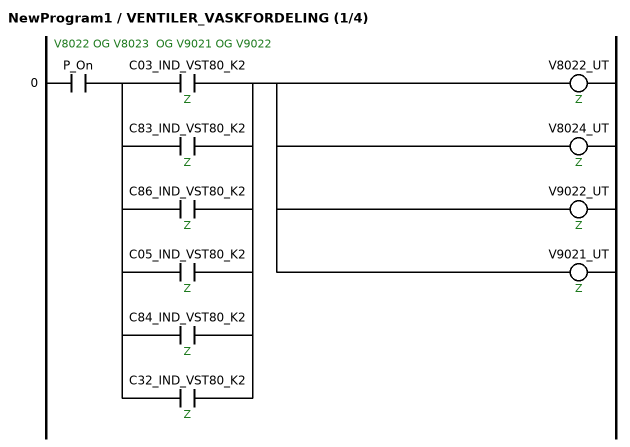
; [picture p840: NewProgram1 / VENTILER_VASKFORDELING, rungs 0-0]
; rung 0: V8022 OG V8023  OG V9021 OG V9022
LD P_On
LD C03_IND_VST80_K2  ; Z
OR C83_IND_VST80_K2  ; Z
OR C86_IND_VST80_K2  ; Z
OR C05_IND_VST80_K2  ; Z
OR C84_IND_VST80_K2  ; Z
OR C32_IND_VST80_K2  ; Z
ANDLD
OUT V8022_UT  ; Z
OUT V8024_UT  ; Z
OUT V9022_UT  ; Z
OUT V9021_UT  ; Z

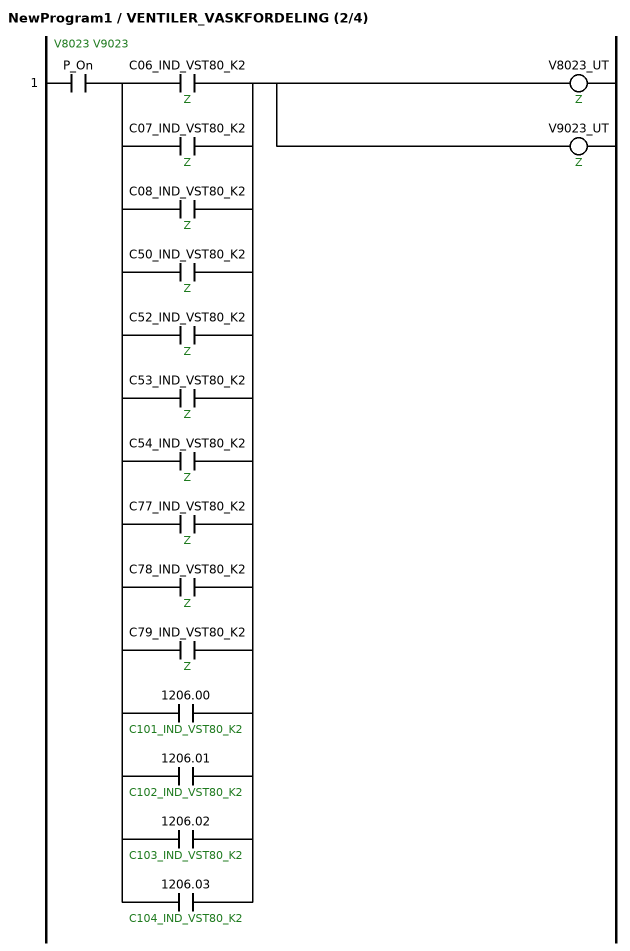
; rung 1: V8023 V9023
LD P_On
LD C06_IND_VST80_K2  ; Z
OR C07_IND_VST80_K2  ; Z
OR C08_IND_VST80_K2  ; Z
OR C50_IND_VST80_K2  ; Z
OR C52_IND_VST80_K2  ; Z
OR C53_IND_VST80_K2  ; Z
OR C54_IND_VST80_K2  ; Z
OR C77_IND_VST80_K2  ; Z
OR C78_IND_VST80_K2  ; Z
OR C79_IND_VST80_K2  ; Z
OR 1206.00  ; C101_IND_VST80_K2
OR 1206.01  ; C102_IND_VST80_K2
OR 1206.02  ; C103_IND_VST80_K2
OR 1206.03  ; C104_IND_VST80_K2
ANDLD
OUT V8023_UT  ; Z
OUT V9023_UT  ; Z

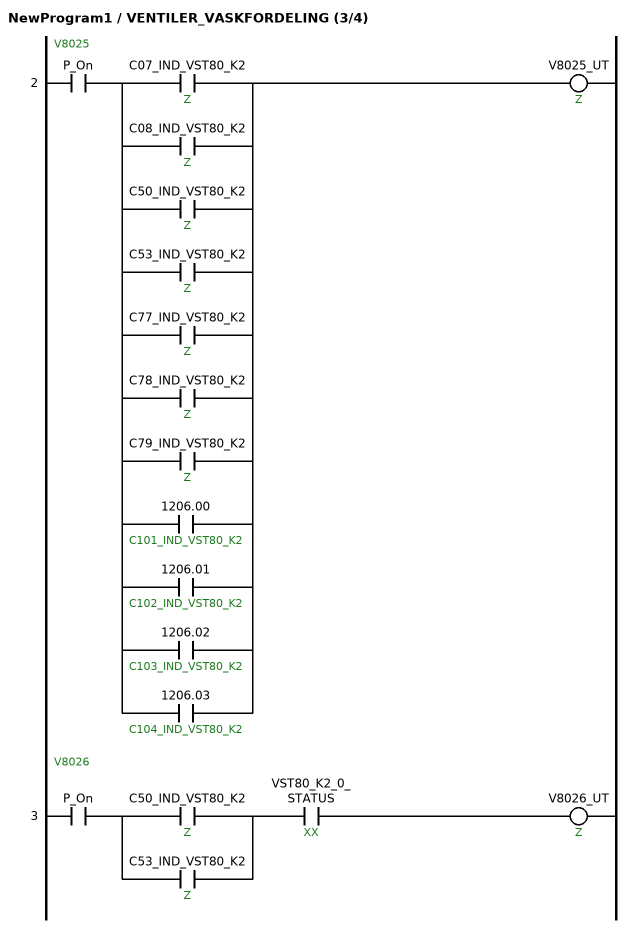
; rung 2: V8025
LD P_On
LD C07_IND_VST80_K2  ; Z
OR C08_IND_VST80_K2  ; Z
OR C50_IND_VST80_K2  ; Z
OR C53_IND_VST80_K2  ; Z
OR C77_IND_VST80_K2  ; Z
OR C78_IND_VST80_K2  ; Z
OR C79_IND_VST80_K2  ; Z
OR 1206.00  ; C101_IND_VST80_K2
OR 1206.01  ; C102_IND_VST80_K2
OR 1206.02  ; C103_IND_VST80_K2
OR 1206.03  ; C104_IND_VST80_K2
ANDLD
OUT V8025_UT  ; Z
; rung 3: V8026
LD P_On
LD C50_IND_VST80_K2  ; Z
OR C53_IND_VST80_K2  ; Z
ANDLD
AND VST80_K2_0_STATUS  ; XX
OUT V8026_UT  ; Z

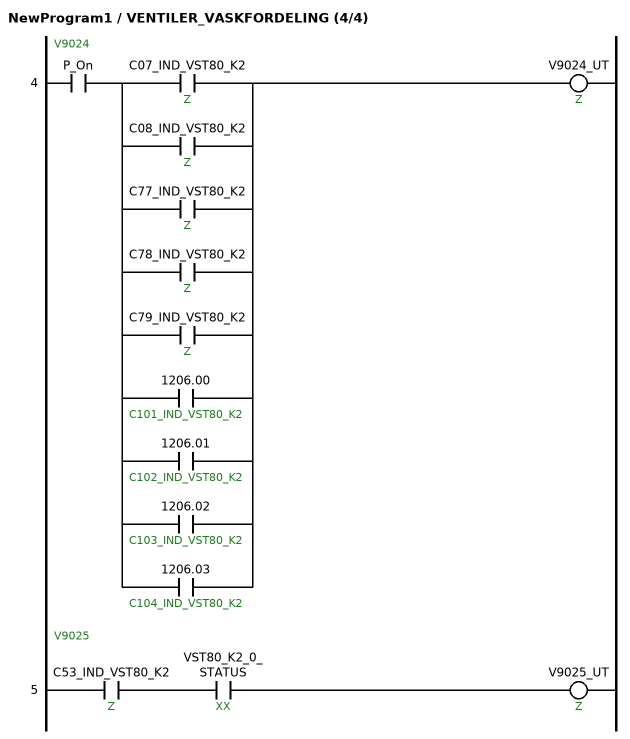
; rung 4: V9024
LD P_On
LD C07_IND_VST80_K2  ; Z
OR C08_IND_VST80_K2  ; Z
OR C77_IND_VST80_K2  ; Z
OR C78_IND_VST80_K2  ; Z
OR C79_IND_VST80_K2  ; Z
OR 1206.00  ; C101_IND_VST80_K2
OR 1206.01  ; C102_IND_VST80_K2
OR 1206.02  ; C103_IND_VST80_K2
OR 1206.03  ; C104_IND_VST80_K2
ANDLD
OUT V9024_UT  ; Z
; rung 5: V9025
LD C53_IND_VST80_K2  ; Z
AND VST80_K2_0_STATUS  ; XX
OUT V9025_UT  ; Z
; rung 6: Ingen_kommentar_funnet

### Section VENTILER_BILVASK

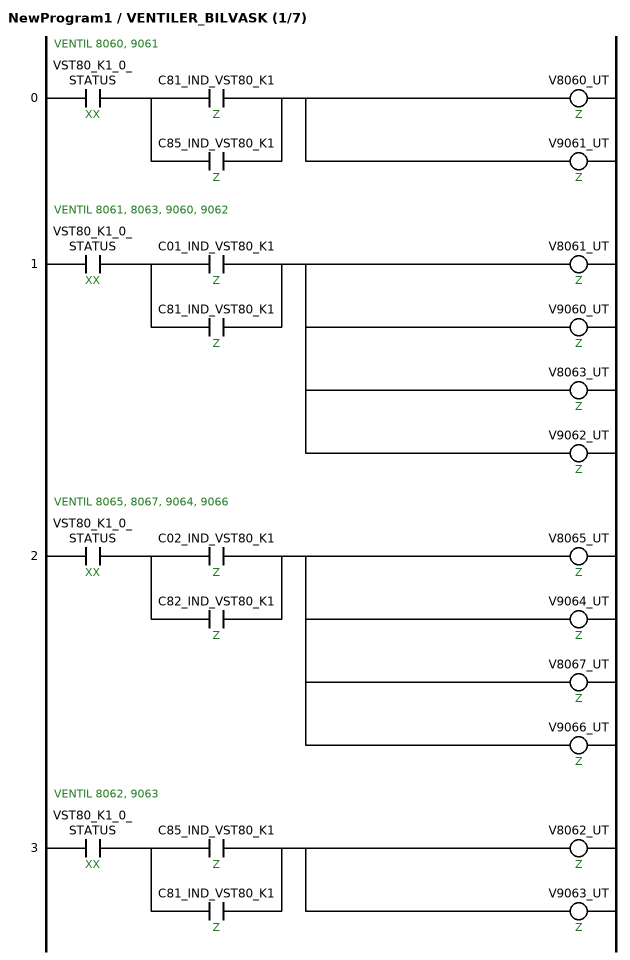
; rung 0: VENTIL 8060, 9061
LD VST80_K1_0_STATUS  ; XX
LD C81_IND_VST80_K1  ; Z
OR C85_IND_VST80_K1  ; Z
ANDLD
OUT V8060_UT  ; Z
OUT V9061_UT  ; Z
; rung 1: VENTIL 8061, 8063, 9060, 9062
LD VST80_K1_0_STATUS  ; XX
LD C01_IND_VST80_K1  ; Z
OR C81_IND_VST80_K1  ; Z
ANDLD
OUT V8061_UT  ; Z
OUT V9060_UT  ; Z
OUT V8063_UT  ; Z
OUT V9062_UT  ; Z
; rung 2: VENTIL 8065, 8067, 9064, 9066
LD VST80_K1_0_STATUS  ; XX
LD C02_IND_VST80_K1  ; Z
OR C82_IND_VST80_K1  ; Z
ANDLD
OUT V8065_UT  ; Z
OUT V9064_UT  ; Z
OUT V8067_UT  ; Z
OUT V9066_UT  ; Z
; rung 3: VENTIL 8062, 9063
LD VST80_K1_0_STATUS  ; XX
LD C85_IND_VST80_K1  ; Z
OR C81_IND_VST80_K1  ; Z
ANDLD
OUT V8062_UT  ; Z
OUT V9063_UT  ; Z

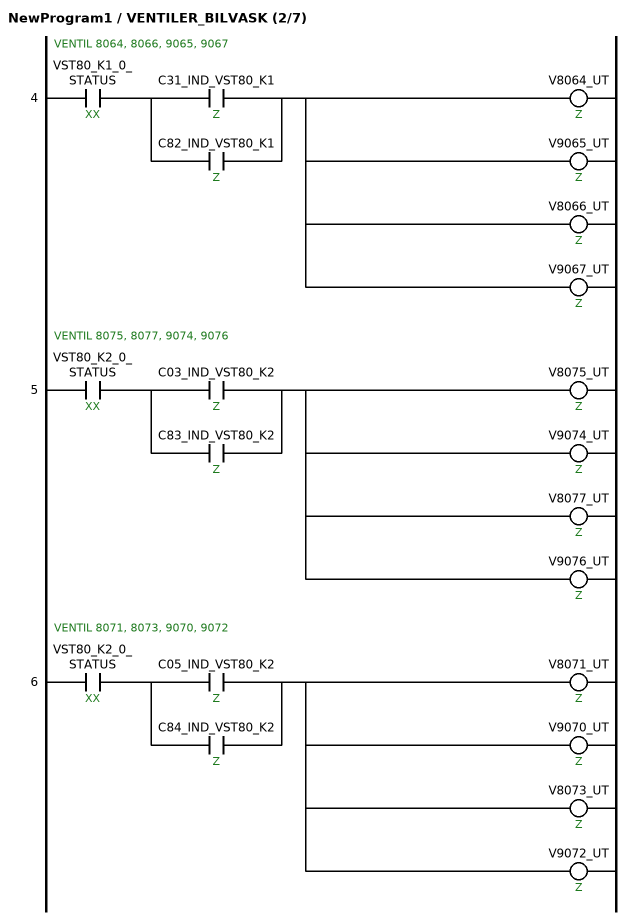
; rung 4: VENTIL 8064, 8066, 9065, 9067
LD VST80_K1_0_STATUS  ; XX
LD C31_IND_VST80_K1  ; Z
OR C82_IND_VST80_K1  ; Z
ANDLD
OUT V8064_UT  ; Z
OUT V9065_UT  ; Z
OUT V8066_UT  ; Z
OUT V9067_UT  ; Z
; rung 5: VENTIL 8075, 8077, 9074, 9076
LD VST80_K2_0_STATUS  ; XX
LD C03_IND_VST80_K2  ; Z
OR C83_IND_VST80_K2  ; Z
ANDLD
OUT V8075_UT  ; Z
OUT V9074_UT  ; Z
OUT V8077_UT  ; Z
OUT V9076_UT  ; Z
; rung 6: VENTIL 8071, 8073, 9070, 9072
LD VST80_K2_0_STATUS  ; XX
LD C05_IND_VST80_K2  ; Z
OR C84_IND_VST80_K2  ; Z
ANDLD
OUT V8071_UT  ; Z
OUT V9070_UT  ; Z
OUT V8073_UT  ; Z
OUT V9072_UT  ; Z

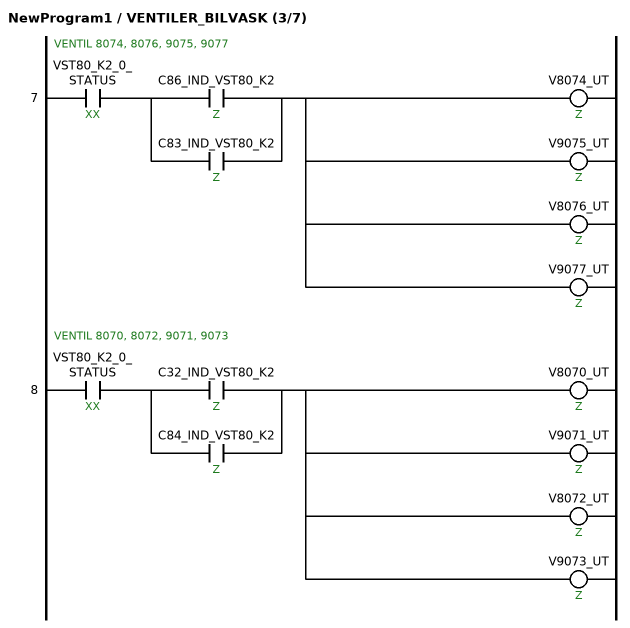
; rung 7: VENTIL 8074, 8076, 9075, 9077
LD VST80_K2_0_STATUS  ; XX
LD C86_IND_VST80_K2  ; Z
OR C83_IND_VST80_K2  ; Z
ANDLD
OUT V8074_UT  ; Z
OUT V9075_UT  ; Z
OUT V8076_UT  ; Z
OUT V9077_UT  ; Z
; rung 8: VENTIL 8070, 8072, 9071, 9073
LD VST80_K2_0_STATUS  ; XX
LD C32_IND_VST80_K2  ; Z
OR C84_IND_VST80_K2  ; Z
ANDLD
OUT V8070_UT  ; Z
OUT V9071_UT  ; Z
OUT V8072_UT  ; Z
OUT V9073_UT  ; Z

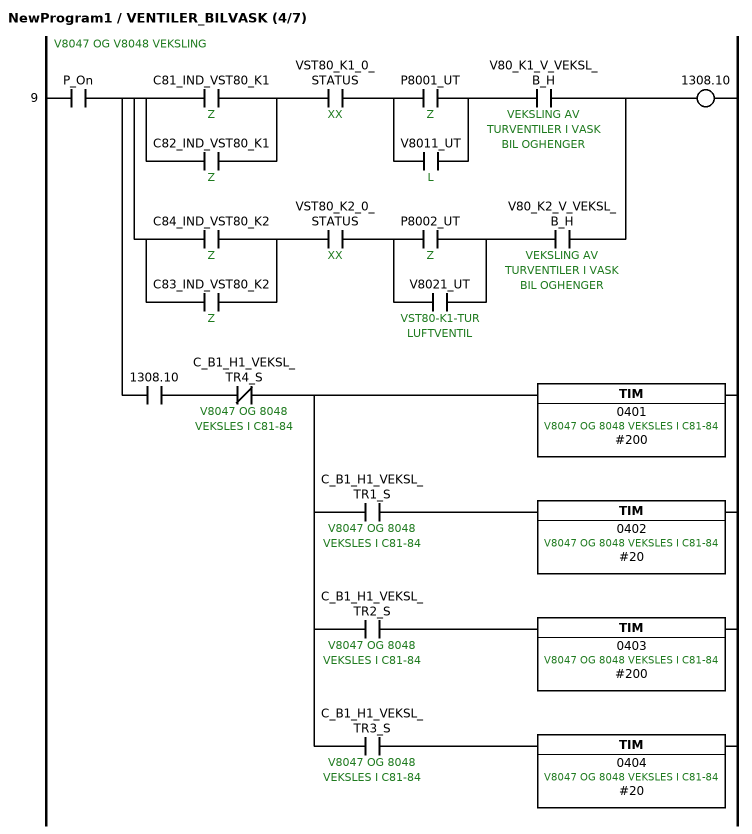
; rung 9: V8047 OG V8048 VEKSLING
LD P_On
OUT TR0
LD C81_IND_VST80_K1  ; Z
OR C82_IND_VST80_K1  ; Z
AND VST80_K1_0_STATUS  ; XX
LD P8001_UT  ; Z
OR V8011_UT  ; L
ANDLD
AND V80_K1_V_VEKSL_B_H  ; VEKSLING AV TURVENTILER I VASK BIL OGHENGER
LD C84_IND_VST80_K2  ; Z
OR C83_IND_VST80_K2  ; Z
AND VST80_K2_0_STATUS  ; XX
LD P8002_UT  ; Z
OR V8021_UT  ; VST80-K1-TUR LUFTVENTIL
ANDLD
AND V80_K2_V_VEKSL_B_H  ; VEKSLING AV TURVENTILER I VASK BIL OGHENGER
ORLD
ANDLD
OUT 1308.10
LD TR0
AND 1308.10
ANDNOT C_B1_H1_VEKSL_TR4_S  ; V8047 OG 8048 VEKSLES I C81-84
OUT TR0
TIM 0401 #200  ; V8047 OG 8048 VEKSLES I C81-84
AND C_B1_H1_VEKSL_TR1_S  ; V8047 OG 8048 VEKSLES I C81-84
TIM 0402 #20  ; V8047 OG 8048 VEKSLES I C81-84
LD TR0
AND C_B1_H1_VEKSL_TR2_S  ; V8047 OG 8048 VEKSLES I C81-84
TIM 0403 #200  ; V8047 OG 8048 VEKSLES I C81-84
LD TR0
AND C_B1_H1_VEKSL_TR3_S  ; V8047 OG 8048 VEKSLES I C81-84
TIM 0404 #20  ; V8047 OG 8048 VEKSLES I C81-84

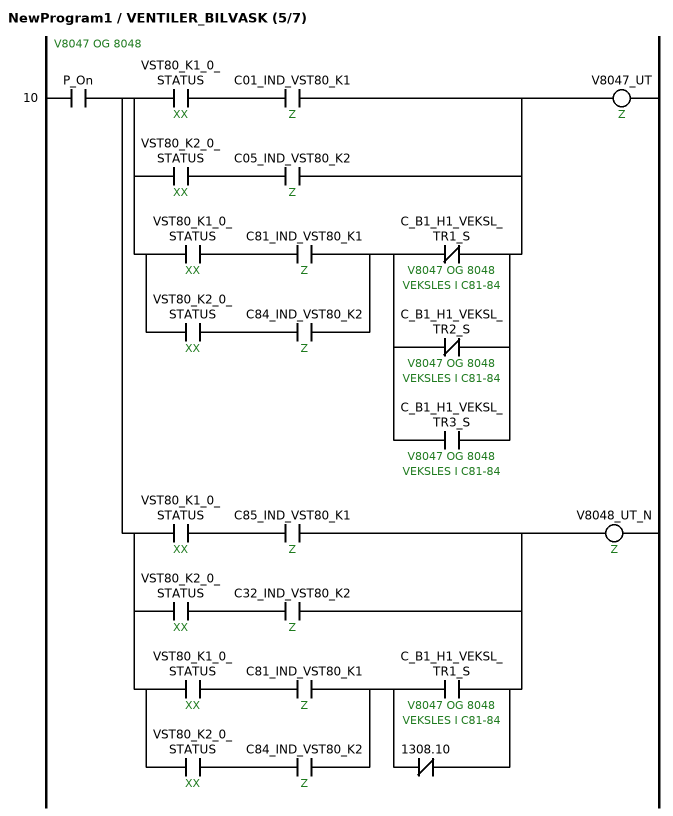
; rung 10: V8047 OG 8048
LD P_On
OUT TR0
LD VST80_K1_0_STATUS  ; XX
AND C01_IND_VST80_K1  ; Z
LD VST80_K2_0_STATUS  ; XX
AND C05_IND_VST80_K2  ; Z
ORLD
LD VST80_K1_0_STATUS  ; XX
AND C81_IND_VST80_K1  ; Z
LD VST80_K2_0_STATUS  ; XX
AND C84_IND_VST80_K2  ; Z
ORLD
LDNOT C_B1_H1_VEKSL_TR1_S  ; V8047 OG 8048 VEKSLES I C81-84
ORNOT C_B1_H1_VEKSL_TR2_S  ; V8047 OG 8048 VEKSLES I C81-84
OR C_B1_H1_VEKSL_TR3_S  ; V8047 OG 8048 VEKSLES I C81-84
ANDLD
ORLD
ANDLD
OUT V8047_UT  ; Z
LD TR0
LD VST80_K1_0_STATUS  ; XX
AND C85_IND_VST80_K1  ; Z
LD VST80_K2_0_STATUS  ; XX
AND C32_IND_VST80_K2  ; Z
ORLD
LD VST80_K1_0_STATUS  ; XX
AND C81_IND_VST80_K1  ; Z
LD VST80_K2_0_STATUS  ; XX
AND C84_IND_VST80_K2  ; Z
ORLD
LD C_B1_H1_VEKSL_TR1_S  ; V8047 OG 8048 VEKSLES I C81-84
ORNOT 1308.10
ANDLD
ORLD
ANDLD
OUT V8048_UT_N  ; Z

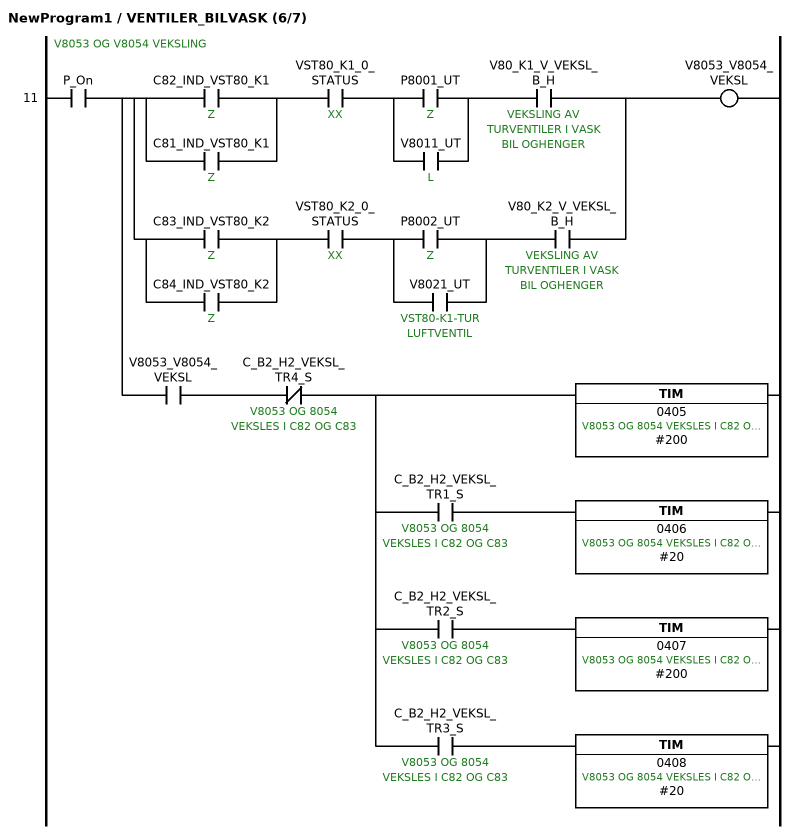
; rung 11: V8053 OG V8054 VEKSLING
LD P_On
OUT TR0
LD C82_IND_VST80_K1  ; Z
OR C81_IND_VST80_K1  ; Z
AND VST80_K1_0_STATUS  ; XX
LD P8001_UT  ; Z
OR V8011_UT  ; L
ANDLD
AND V80_K1_V_VEKSL_B_H  ; VEKSLING AV TURVENTILER I VASK BIL OGHENGER
LD C83_IND_VST80_K2  ; Z
OR C84_IND_VST80_K2  ; Z
AND VST80_K2_0_STATUS  ; XX
LD P8002_UT  ; Z
OR V8021_UT  ; VST80-K1-TUR LUFTVENTIL
ANDLD
AND V80_K2_V_VEKSL_B_H  ; VEKSLING AV TURVENTILER I VASK BIL OGHENGER
ORLD
ANDLD
OUT V8053_V8054_VEKSL
LD TR0
AND V8053_V8054_VEKSL
ANDNOT C_B2_H2_VEKSL_TR4_S  ; V8053 OG 8054 VEKSLES I C82 OG C83
OUT TR0
TIM 0405 #200  ; V8053 OG 8054 VEKSLES I C82 OG C83
AND C_B2_H2_VEKSL_TR1_S  ; V8053 OG 8054 VEKSLES I C82 OG C83
TIM 0406 #20  ; V8053 OG 8054 VEKSLES I C82 OG C83
LD TR0
AND C_B2_H2_VEKSL_TR2_S  ; V8053 OG 8054 VEKSLES I C82 OG C83
TIM 0407 #200  ; V8053 OG 8054 VEKSLES I C82 OG C83
LD TR0
AND C_B2_H2_VEKSL_TR3_S  ; V8053 OG 8054 VEKSLES I C82 OG C83
TIM 0408 #20  ; V8053 OG 8054 VEKSLES I C82 OG C83

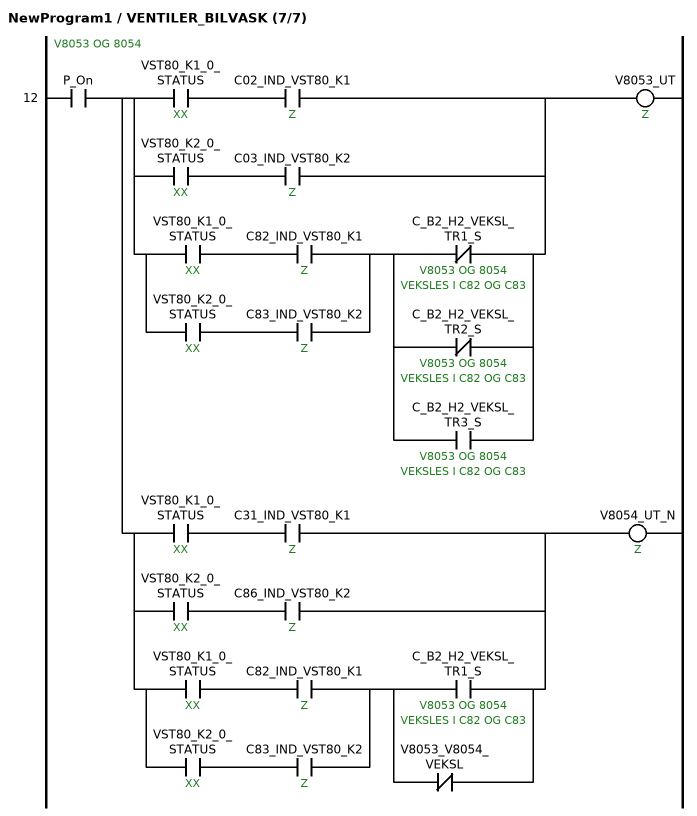
; rung 12: V8053 OG 8054
LD P_On
OUT TR0
LD VST80_K1_0_STATUS  ; XX
AND C02_IND_VST80_K1  ; Z
LD VST80_K2_0_STATUS  ; XX
AND C03_IND_VST80_K2  ; Z
ORLD
LD VST80_K1_0_STATUS  ; XX
AND C82_IND_VST80_K1  ; Z
LD VST80_K2_0_STATUS  ; XX
AND C83_IND_VST80_K2  ; Z
ORLD
LDNOT C_B2_H2_VEKSL_TR1_S  ; V8053 OG 8054 VEKSLES I C82 OG C83
ORNOT C_B2_H2_VEKSL_TR2_S  ; V8053 OG 8054 VEKSLES I C82 OG C83
OR C_B2_H2_VEKSL_TR3_S  ; V8053 OG 8054 VEKSLES I C82 OG C83
ANDLD
ORLD
ANDLD
OUT V8053_UT  ; Z
LD TR0
LD VST80_K1_0_STATUS  ; XX
AND C31_IND_VST80_K1  ; Z
LD VST80_K2_0_STATUS  ; XX
AND C86_IND_VST80_K2  ; Z
ORLD
LD VST80_K1_0_STATUS  ; XX
AND C82_IND_VST80_K1  ; Z
LD VST80_K2_0_STATUS  ; XX
AND C83_IND_VST80_K2  ; Z
ORLD
LD C_B2_H2_VEKSL_TR1_S  ; V8053 OG 8054 VEKSLES I C82 OG C83
ORNOT V8053_V8054_VEKSL
ANDLD
ORLD
ANDLD
OUT V8054_UT_N  ; Z
; rung 13: Ingen_kommentar_funnet

### Section VENTILER_SILOTANKER

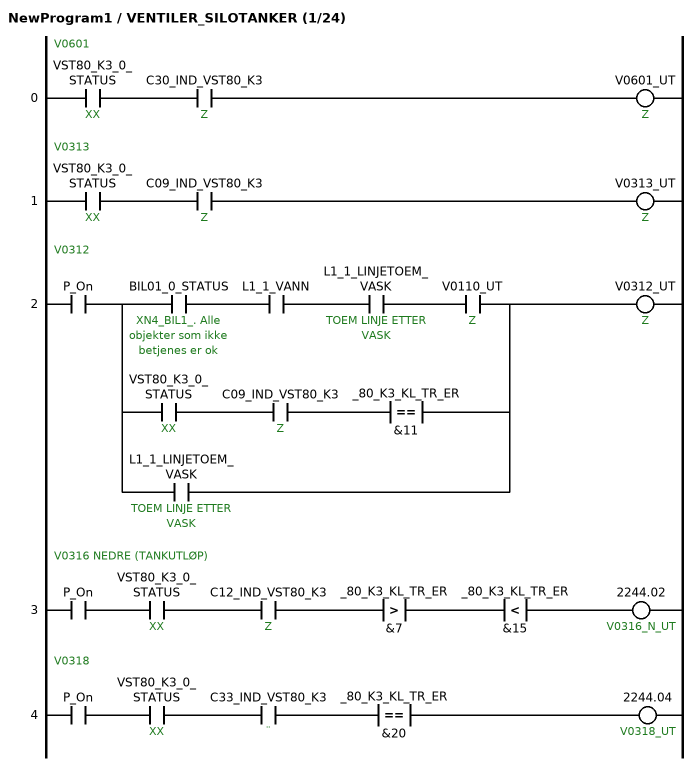
; rung 0: V0601
LD VST80_K3_0_STATUS  ; XX
AND C30_IND_VST80_K3  ; Z
OUT V0601_UT  ; Z
; rung 1: V0313
LD VST80_K3_0_STATUS  ; XX
AND C09_IND_VST80_K3  ; Z
OUT V0313_UT  ; Z
; rung 2: V0312
LD P_On
LD BIL01_0_STATUS  ; XN4_BIL1_. Alle objekter som ikke betjenes er ok
AND L1_1_VANN
AND L1_1_LINJETOEM_VASK  ; TOEM LINJE ETTER VASK
AND V0110_UT  ; Z
LD VST80_K3_0_STATUS  ; XX
AND C09_IND_VST80_K3  ; Z
AND=(300) _80_K3_KL_TR_ER &11
ORLD
OR L1_1_LINJETOEM_VASK  ; TOEM LINJE ETTER VASK
ANDLD
OUT V0312_UT  ; Z
; rung 3: V0316 NEDRE (TANKUTLØP)
LD P_On
AND VST80_K3_0_STATUS  ; XX
AND C12_IND_VST80_K3  ; Z
AND>(320) _80_K3_KL_TR_ER &7
AND<(310) _80_K3_KL_TR_ER &15
OUT 2244.02  ; V0316_N_UT
; rung 4: V0318
LD P_On
AND VST80_K3_0_STATUS  ; XX
AND C33_IND_VST80_K3  ; ¨
AND=(300) _80_K3_KL_TR_ER &20
OUT 2244.04  ; V0318_UT

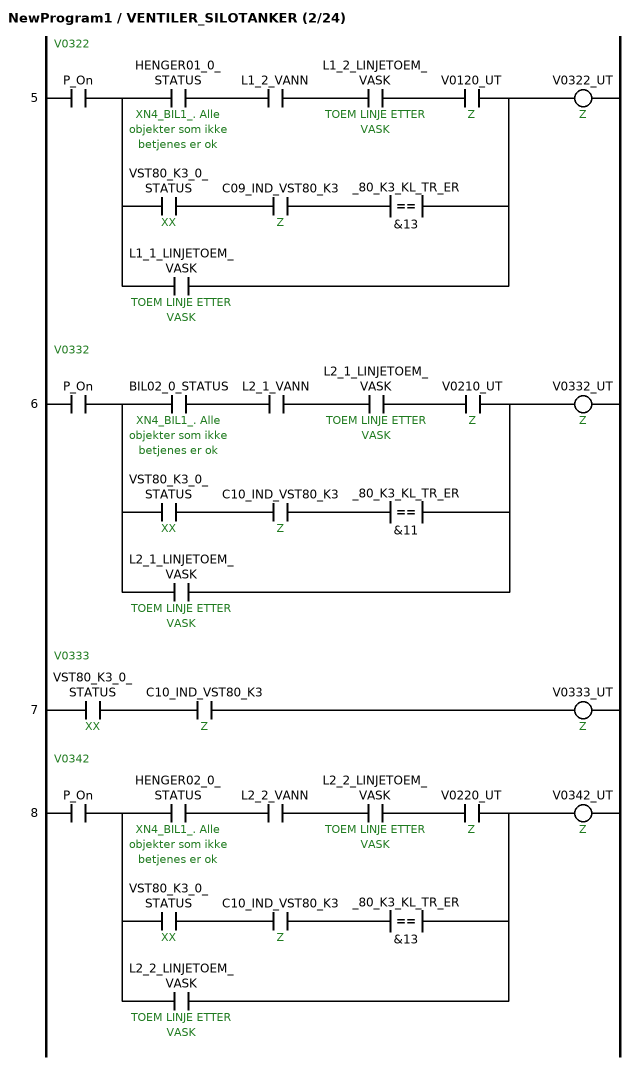
; rung 5: V0322
LD P_On
LD HENGER01_0_STATUS  ; XN4_BIL1_. Alle objekter som ikke betjenes er ok
AND L1_2_VANN
AND L1_2_LINJETOEM_VASK  ; TOEM LINJE ETTER VASK
AND V0120_UT  ; Z
LD VST80_K3_0_STATUS  ; XX
AND C09_IND_VST80_K3  ; Z
AND=(300) _80_K3_KL_TR_ER &13
ORLD
OR L1_1_LINJETOEM_VASK  ; TOEM LINJE ETTER VASK
ANDLD
OUT V0322_UT  ; Z
; rung 6: V0332
LD P_On
LD BIL02_0_STATUS  ; XN4_BIL1_. Alle objekter som ikke betjenes er ok
AND L2_1_VANN
AND L2_1_LINJETOEM_VASK  ; TOEM LINJE ETTER VASK
AND V0210_UT  ; Z
LD VST80_K3_0_STATUS  ; XX
AND C10_IND_VST80_K3  ; Z
AND=(300) _80_K3_KL_TR_ER &11
ORLD
OR L2_1_LINJETOEM_VASK  ; TOEM LINJE ETTER VASK
ANDLD
OUT V0332_UT  ; Z
; rung 7: V0333
LD VST80_K3_0_STATUS  ; XX
AND C10_IND_VST80_K3  ; Z
OUT V0333_UT  ; Z
; rung 8: V0342
LD P_On
LD HENGER02_0_STATUS  ; XN4_BIL1_. Alle objekter som ikke betjenes er ok
AND L2_2_VANN
AND L2_2_LINJETOEM_VASK  ; TOEM LINJE ETTER VASK
AND V0220_UT  ; Z
LD VST80_K3_0_STATUS  ; XX
AND C10_IND_VST80_K3  ; Z
AND=(300) _80_K3_KL_TR_ER &13
ORLD
OR L2_2_LINJETOEM_VASK  ; TOEM LINJE ETTER VASK
ANDLD
OUT V0342_UT  ; Z

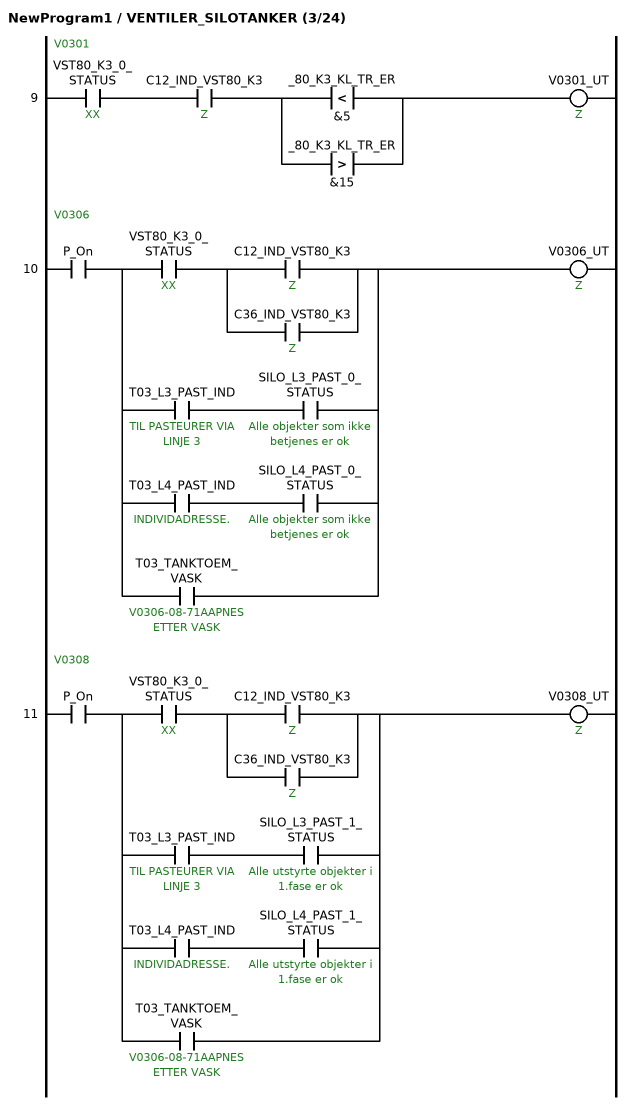
; rung 9: V0301
LD VST80_K3_0_STATUS  ; XX
AND C12_IND_VST80_K3  ; Z
LD<(310) _80_K3_KL_TR_ER &5
OR>(320) _80_K3_KL_TR_ER &15
ANDLD
OUT V0301_UT  ; Z
; rung 10: V0306
LD P_On
LD VST80_K3_0_STATUS  ; XX
LD C12_IND_VST80_K3  ; Z
OR C36_IND_VST80_K3  ; Z
ANDLD
LD T03_L3_PAST_IND  ; TIL PASTEURER VIA LINJE 3
AND SILO_L3_PAST_0_STATUS  ; Alle objekter som ikke betjenes er ok
ORLD
LD T03_L4_PAST_IND  ; INDIVIDADRESSE.
AND SILO_L4_PAST_0_STATUS  ; Alle objekter som ikke betjenes er ok
ORLD
OR T03_TANKTOEM_VASK  ; V0306-08-71AAPNES ETTER VASK
ANDLD
OUT V0306_UT  ; Z
; rung 11: V0308
LD P_On
LD VST80_K3_0_STATUS  ; XX
LD C12_IND_VST80_K3  ; Z
OR C36_IND_VST80_K3  ; Z
ANDLD
LD T03_L3_PAST_IND  ; TIL PASTEURER VIA LINJE 3
AND SILO_L3_PAST_1_STATUS  ; Alle utstyrte objekter i 1.fase er ok
ORLD
LD T03_L4_PAST_IND  ; INDIVIDADRESSE.
AND SILO_L4_PAST_1_STATUS  ; Alle utstyrte objekter i 1.fase er ok
ORLD
OR T03_TANKTOEM_VASK  ; V0306-08-71AAPNES ETTER VASK
ANDLD
OUT V0308_UT  ; Z

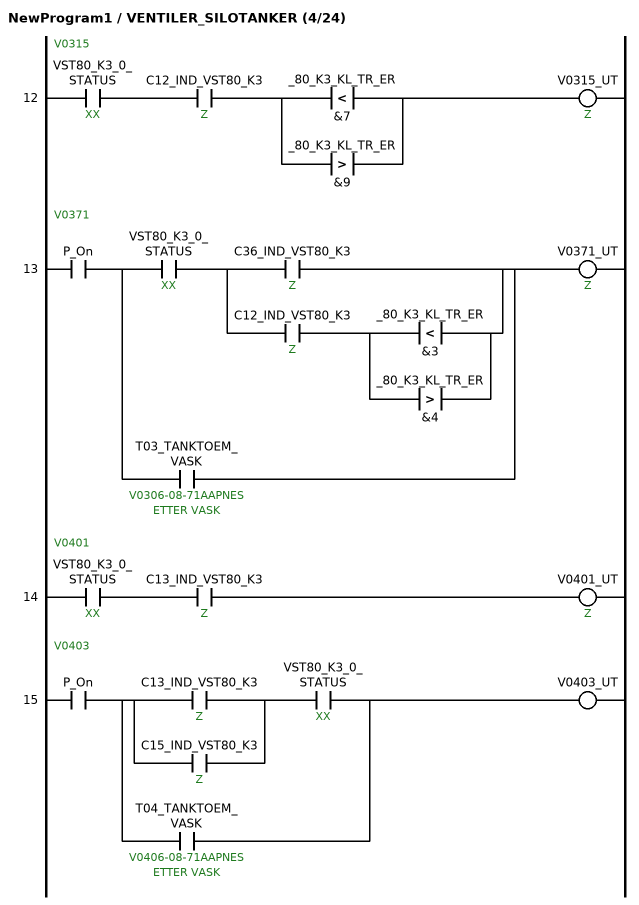
; rung 12: V0315
LD VST80_K3_0_STATUS  ; XX
AND C12_IND_VST80_K3  ; Z
LD<(310) _80_K3_KL_TR_ER &7
OR>(320) _80_K3_KL_TR_ER &9
ANDLD
OUT V0315_UT  ; Z
; rung 13: V0371
LD P_On
LD VST80_K3_0_STATUS  ; XX
LD C36_IND_VST80_K3  ; Z
LD C12_IND_VST80_K3  ; Z
LD<(310) _80_K3_KL_TR_ER &3
OR>(320) _80_K3_KL_TR_ER &4
ANDLD
ORLD
ANDLD
OR T03_TANKTOEM_VASK  ; V0306-08-71AAPNES ETTER VASK
ANDLD
OUT V0371_UT  ; Z
; rung 14: V0401
LD VST80_K3_0_STATUS  ; XX
AND C13_IND_VST80_K3  ; Z
OUT V0401_UT  ; Z
; rung 15: V0403
LD P_On
LD C13_IND_VST80_K3  ; Z
OR C15_IND_VST80_K3  ; Z
AND VST80_K3_0_STATUS  ; XX
OR T04_TANKTOEM_VASK  ; V0406-08-71AAPNES ETTER VASK
ANDLD
OUT V0403_UT

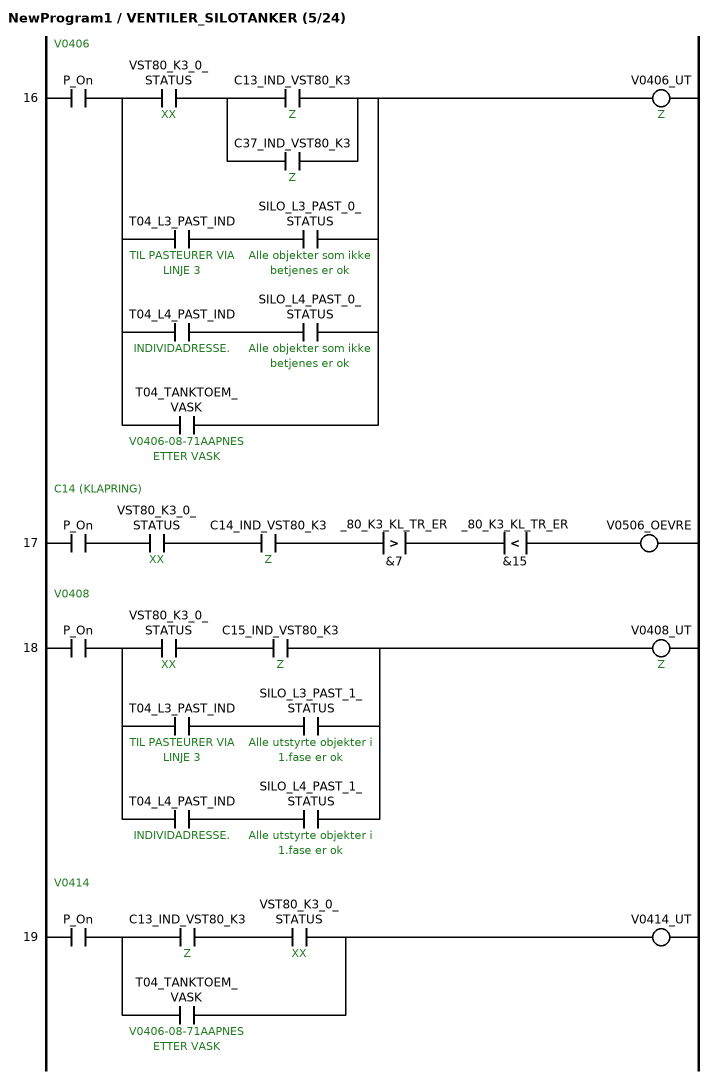
; rung 16: V0406
LD P_On
LD VST80_K3_0_STATUS  ; XX
LD C13_IND_VST80_K3  ; Z
OR C37_IND_VST80_K3  ; Z
ANDLD
LD T04_L3_PAST_IND  ; TIL PASTEURER VIA LINJE 3
AND SILO_L3_PAST_0_STATUS  ; Alle objekter som ikke betjenes er ok
ORLD
LD T04_L4_PAST_IND  ; INDIVIDADRESSE.
AND SILO_L4_PAST_0_STATUS  ; Alle objekter som ikke betjenes er ok
ORLD
OR T04_TANKTOEM_VASK  ; V0406-08-71AAPNES ETTER VASK
ANDLD
OUT V0406_UT  ; Z
; rung 17: C14 (KLAPRING)
LD P_On
AND VST80_K3_0_STATUS  ; XX
AND C14_IND_VST80_K3  ; Z
AND>(320) _80_K3_KL_TR_ER &7
AND<(310) _80_K3_KL_TR_ER &15
OUT V0506_OEVRE
; rung 18: V0408
LD P_On
LD VST80_K3_0_STATUS  ; XX
AND C15_IND_VST80_K3  ; Z
LD T04_L3_PAST_IND  ; TIL PASTEURER VIA LINJE 3
AND SILO_L3_PAST_1_STATUS  ; Alle utstyrte objekter i 1.fase er ok
ORLD
LD T04_L4_PAST_IND  ; INDIVIDADRESSE.
AND SILO_L4_PAST_1_STATUS  ; Alle utstyrte objekter i 1.fase er ok
ORLD
ANDLD
OUT V0408_UT  ; Z
; rung 19: V0414
LD P_On
LD C13_IND_VST80_K3  ; Z
AND VST80_K3_0_STATUS  ; XX
OR T04_TANKTOEM_VASK  ; V0406-08-71AAPNES ETTER VASK
ANDLD
OUT V0414_UT

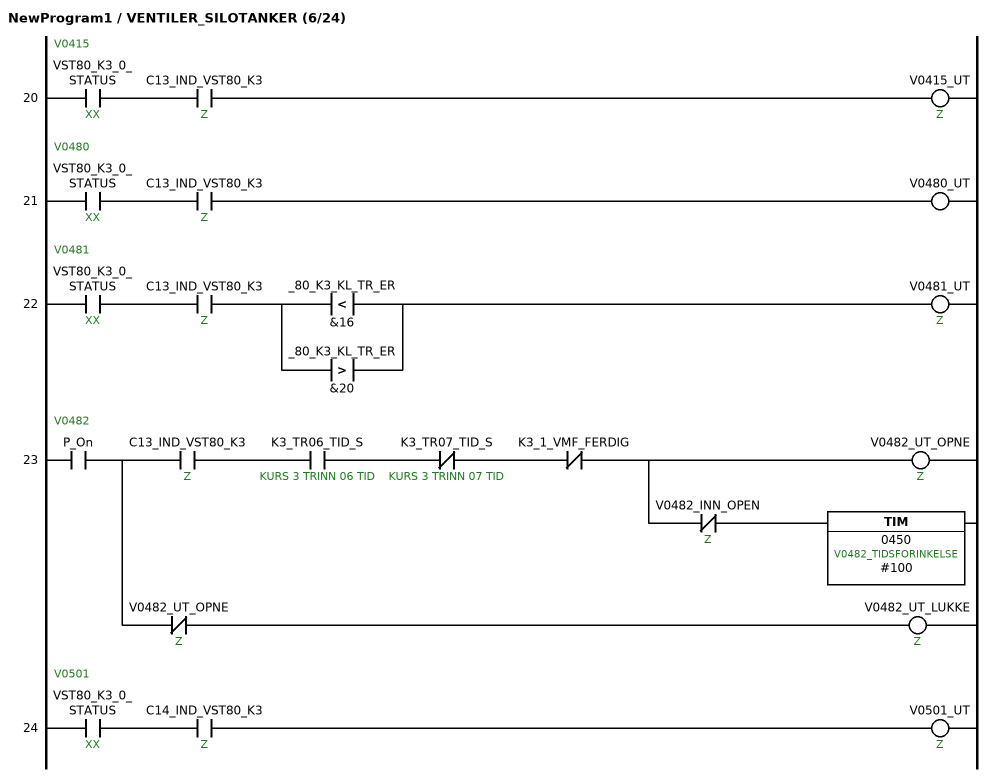
; rung 20: V0415
LD VST80_K3_0_STATUS  ; XX
AND C13_IND_VST80_K3  ; Z
OUT V0415_UT  ; Z
; rung 21: V0480
LD VST80_K3_0_STATUS  ; XX
AND C13_IND_VST80_K3  ; Z
OUT V0480_UT
; rung 22: V0481
LD VST80_K3_0_STATUS  ; XX
AND C13_IND_VST80_K3  ; Z
LD<(310) _80_K3_KL_TR_ER &16
OR>(320) _80_K3_KL_TR_ER &20
ANDLD
OUT V0481_UT  ; Z
; rung 23: V0482
LD P_On
OUT TR0
AND C13_IND_VST80_K3  ; Z
AND K3_TR06_TID_S  ; KURS 3 TRINN 06 TID
ANDNOT K3_TR07_TID_S  ; KURS 3 TRINN 07 TID
ANDNOT K3_1_VMF_FERDIG
OUT V0482_UT_OPNE  ; Z
ANDNOT V0482_INN_OPEN  ; Z
TIM 0450 #100  ; V0482_TIDSFORINKELSE
LD TR0
ANDNOT V0482_UT_OPNE  ; Z
OUT V0482_UT_LUKKE  ; Z
; rung 24: V0501
LD VST80_K3_0_STATUS  ; XX
AND C14_IND_VST80_K3  ; Z
OUT V0501_UT  ; Z

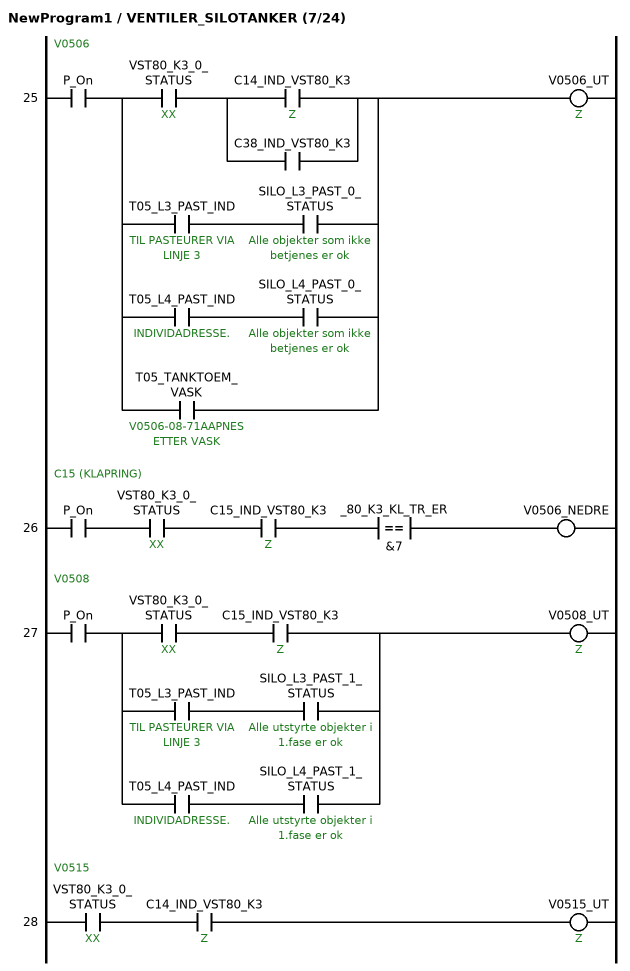
; rung 25: V0506
LD P_On
LD VST80_K3_0_STATUS  ; XX
LD C14_IND_VST80_K3  ; Z
OR C38_IND_VST80_K3
ANDLD
LD T05_L3_PAST_IND  ; TIL PASTEURER VIA LINJE 3
AND SILO_L3_PAST_0_STATUS  ; Alle objekter som ikke betjenes er ok
ORLD
LD T05_L4_PAST_IND  ; INDIVIDADRESSE.
AND SILO_L4_PAST_0_STATUS  ; Alle objekter som ikke betjenes er ok
ORLD
OR T05_TANKTOEM_VASK  ; V0506-08-71AAPNES ETTER VASK
ANDLD
OUT V0506_UT  ; Z
; rung 26: C15 (KLAPRING)
LD P_On
AND VST80_K3_0_STATUS  ; XX
AND C15_IND_VST80_K3  ; Z
AND=(300) _80_K3_KL_TR_ER &7
OUT V0506_NEDRE
; rung 27: V0508
LD P_On
LD VST80_K3_0_STATUS  ; XX
AND C15_IND_VST80_K3  ; Z
LD T05_L3_PAST_IND  ; TIL PASTEURER VIA LINJE 3
AND SILO_L3_PAST_1_STATUS  ; Alle utstyrte objekter i 1.fase er ok
ORLD
LD T05_L4_PAST_IND  ; INDIVIDADRESSE.
AND SILO_L4_PAST_1_STATUS  ; Alle utstyrte objekter i 1.fase er ok
ORLD
ANDLD
OUT V0508_UT  ; Z
; rung 28: V0515
LD VST80_K3_0_STATUS  ; XX
AND C14_IND_VST80_K3  ; Z
OUT V0515_UT  ; Z

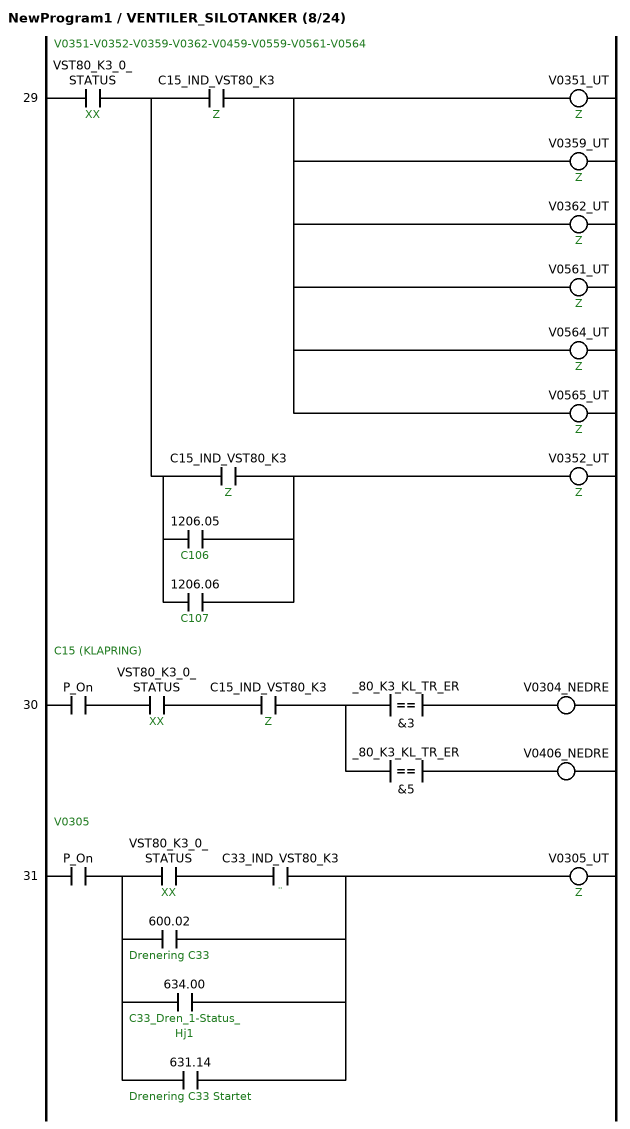
; rung 29: V0351-V0352-V0359-V0362-V0459-V0559-V0561-V0564
LD VST80_K3_0_STATUS  ; XX
OUT TR0
AND C15_IND_VST80_K3  ; Z
OUT V0351_UT  ; Z
OUT V0359_UT  ; Z
OUT V0362_UT  ; Z
OUT V0561_UT  ; Z
OUT V0564_UT  ; Z
OUT V0565_UT  ; Z
LD TR0
LD C15_IND_VST80_K3  ; Z
OR 1206.05  ; C106
OR 1206.06  ; C107
ANDLD
OUT V0352_UT  ; Z
; rung 30: C15 (KLAPRING)
LD P_On
AND VST80_K3_0_STATUS  ; XX
AND C15_IND_VST80_K3  ; Z
OUT TR0
AND=(300) _80_K3_KL_TR_ER &3
OUT V0304_NEDRE
LD TR0
AND=(300) _80_K3_KL_TR_ER &5
OUT V0406_NEDRE
; rung 31: V0305
LD P_On
LD VST80_K3_0_STATUS  ; XX
AND C33_IND_VST80_K3  ; ¨
OR 600.02  ; Drenering C33
OR 634.00  ; C33_Dren_1-Status_Hj1
OR 631.14  ; Drenering C33 Startet
ANDLD
OUT V0305_UT  ; Z

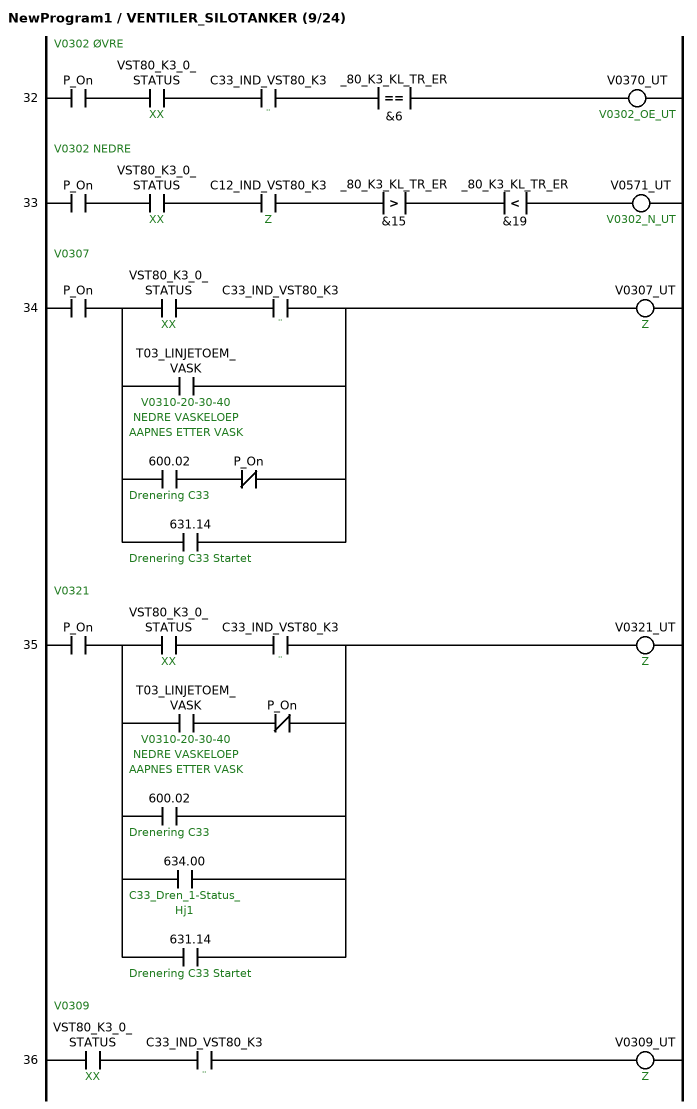
; rung 32: V0302 ØVRE
LD P_On
AND VST80_K3_0_STATUS  ; XX
AND C33_IND_VST80_K3  ; ¨
AND=(300) _80_K3_KL_TR_ER &6
OUT V0370_UT  ; V0302_OE_UT
; rung 33: V0302 NEDRE
LD P_On
AND VST80_K3_0_STATUS  ; XX
AND C12_IND_VST80_K3  ; Z
AND>(320) _80_K3_KL_TR_ER &15
AND<(310) _80_K3_KL_TR_ER &19
OUT V0571_UT  ; V0302_N_UT
; rung 34: V0307
LD P_On
LD VST80_K3_0_STATUS  ; XX
AND C33_IND_VST80_K3  ; ¨
OR T03_LINJETOEM_VASK  ; V0310-20-30-40 NEDRE VASKELOEP AAPNES ETTER VASK
LD 600.02  ; Drenering C33
ANDNOT P_On
ORLD
OR 631.14  ; Drenering C33 Startet
ANDLD
OUT V0307_UT  ; Z
; rung 35: V0321
LD P_On
LD VST80_K3_0_STATUS  ; XX
AND C33_IND_VST80_K3  ; ¨
LD T03_LINJETOEM_VASK  ; V0310-20-30-40 NEDRE VASKELOEP AAPNES ETTER VASK
ANDNOT P_On
ORLD
OR 600.02  ; Drenering C33
OR 634.00  ; C33_Dren_1-Status_Hj1
OR 631.14  ; Drenering C33 Startet
ANDLD
OUT V0321_UT  ; Z
; rung 36: V0309
LD VST80_K3_0_STATUS  ; XX
AND C33_IND_VST80_K3  ; ¨
OUT V0309_UT  ; Z

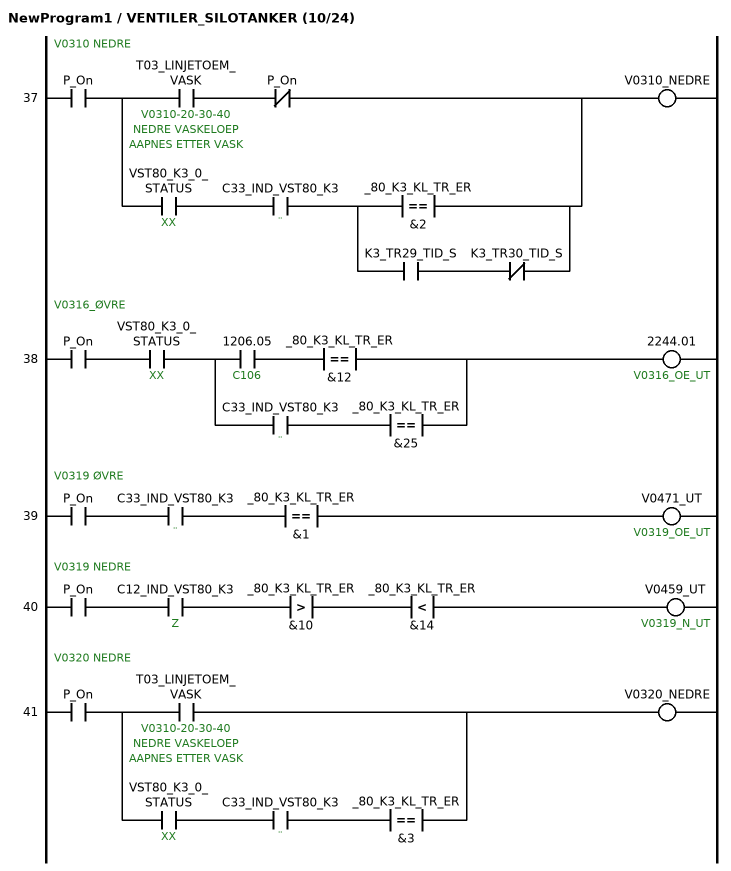
; rung 37: V0310 NEDRE
LD P_On
LD T03_LINJETOEM_VASK  ; V0310-20-30-40 NEDRE VASKELOEP AAPNES ETTER VASK
ANDNOT P_On
LD VST80_K3_0_STATUS  ; XX
AND C33_IND_VST80_K3  ; ¨
LD=(300) _80_K3_KL_TR_ER &2
LD K3_TR29_TID_S
ANDNOT K3_TR30_TID_S
ORLD
ANDLD
ORLD
ANDLD
OUT V0310_NEDRE
; rung 38: V0316_ØVRE
LD P_On
AND VST80_K3_0_STATUS  ; XX
LD 1206.05  ; C106
AND=(300) _80_K3_KL_TR_ER &12
LD C33_IND_VST80_K3  ; ¨
AND=(300) _80_K3_KL_TR_ER &25
ORLD
ANDLD
OUT 2244.01  ; V0316_OE_UT
; rung 39: V0319 ØVRE
LD P_On
AND C33_IND_VST80_K3  ; ¨
AND=(300) _80_K3_KL_TR_ER &1
OUT V0471_UT  ; V0319_OE_UT
; rung 40: V0319 NEDRE
LD P_On
AND C12_IND_VST80_K3  ; Z
AND>(320) _80_K3_KL_TR_ER &10
AND<(310) _80_K3_KL_TR_ER &14
OUT V0459_UT  ; V0319_N_UT
; rung 41: V0320 NEDRE
LD P_On
LD T03_LINJETOEM_VASK  ; V0310-20-30-40 NEDRE VASKELOEP AAPNES ETTER VASK
LD VST80_K3_0_STATUS  ; XX
AND C33_IND_VST80_K3  ; ¨
AND=(300) _80_K3_KL_TR_ER &3
ORLD
ANDLD
OUT V0320_NEDRE

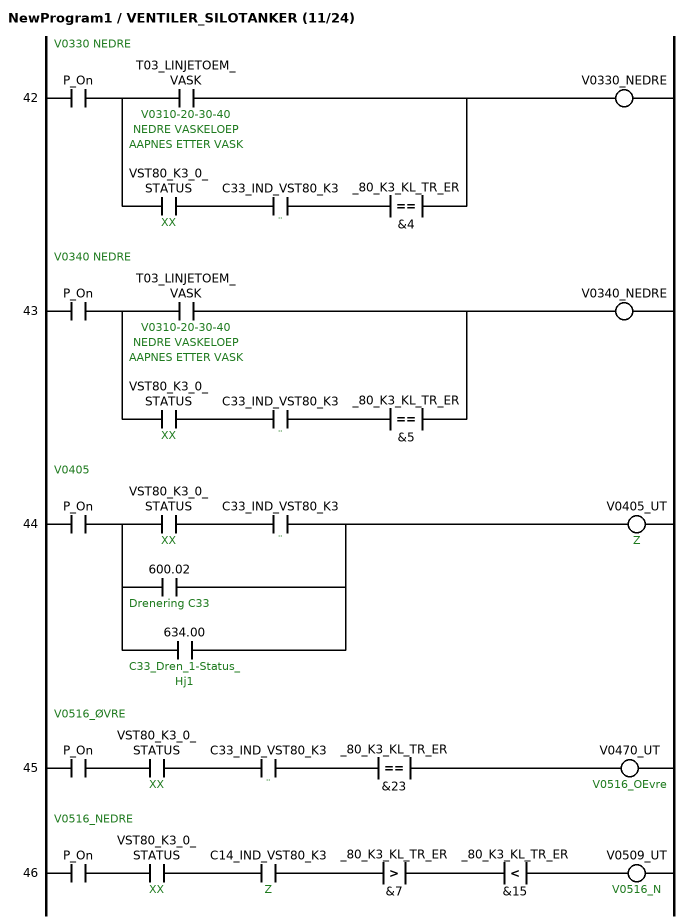
; rung 42: V0330 NEDRE
LD P_On
LD T03_LINJETOEM_VASK  ; V0310-20-30-40 NEDRE VASKELOEP AAPNES ETTER VASK
LD VST80_K3_0_STATUS  ; XX
AND C33_IND_VST80_K3  ; ¨
AND=(300) _80_K3_KL_TR_ER &4
ORLD
ANDLD
OUT V0330_NEDRE
; rung 43: V0340 NEDRE
LD P_On
LD T03_LINJETOEM_VASK  ; V0310-20-30-40 NEDRE VASKELOEP AAPNES ETTER VASK
LD VST80_K3_0_STATUS  ; XX
AND C33_IND_VST80_K3  ; ¨
AND=(300) _80_K3_KL_TR_ER &5
ORLD
ANDLD
OUT V0340_NEDRE
; rung 44: V0405
LD P_On
LD VST80_K3_0_STATUS  ; XX
AND C33_IND_VST80_K3  ; ¨
OR 600.02  ; Drenering C33
OR 634.00  ; C33_Dren_1-Status_Hj1
ANDLD
OUT V0405_UT  ; Z
; rung 45: V0516_ØVRE
LD P_On
AND VST80_K3_0_STATUS  ; XX
AND C33_IND_VST80_K3  ; ¨
AND=(300) _80_K3_KL_TR_ER &23
OUT V0470_UT  ; V0516_OEvre
; rung 46: V0516_NEDRE
LD P_On
AND VST80_K3_0_STATUS  ; XX
AND C14_IND_VST80_K3  ; Z
AND>(320) _80_K3_KL_TR_ER &7
AND<(310) _80_K3_KL_TR_ER &15
OUT V0509_UT  ; V0516_N

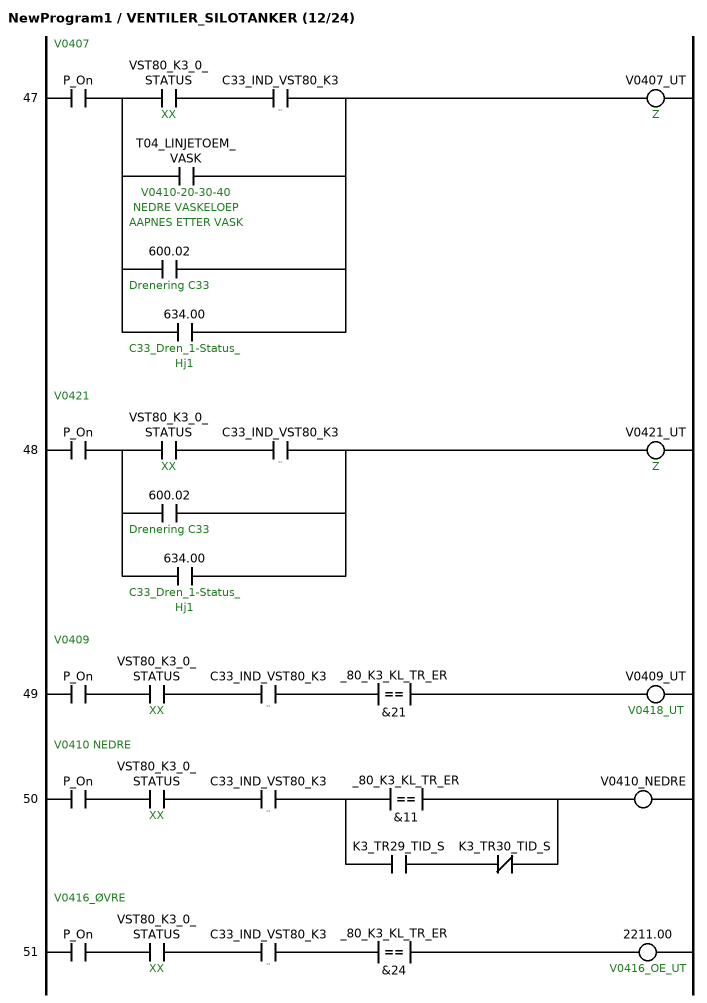
; rung 47: V0407
LD P_On
LD VST80_K3_0_STATUS  ; XX
AND C33_IND_VST80_K3  ; ¨
OR T04_LINJETOEM_VASK  ; V0410-20-30-40 NEDRE VASKELOEP AAPNES ETTER VASK
OR 600.02  ; Drenering C33
OR 634.00  ; C33_Dren_1-Status_Hj1
ANDLD
OUT V0407_UT  ; Z
; rung 48: V0421
LD P_On
LD VST80_K3_0_STATUS  ; XX
AND C33_IND_VST80_K3  ; ¨
OR 600.02  ; Drenering C33
OR 634.00  ; C33_Dren_1-Status_Hj1
ANDLD
OUT V0421_UT  ; Z
; rung 49: V0409
LD P_On
AND VST80_K3_0_STATUS  ; XX
AND C33_IND_VST80_K3  ; ¨
AND=(300) _80_K3_KL_TR_ER &21
OUT V0409_UT  ; V0418_UT
; rung 50: V0410 NEDRE
LD P_On
AND VST80_K3_0_STATUS  ; XX
AND C33_IND_VST80_K3  ; ¨
LD=(300) _80_K3_KL_TR_ER &11
LD K3_TR29_TID_S
ANDNOT K3_TR30_TID_S
ORLD
ANDLD
OUT V0410_NEDRE
; rung 51: V0416_ØVRE
LD P_On
AND VST80_K3_0_STATUS  ; XX
AND C33_IND_VST80_K3  ; ¨
AND=(300) _80_K3_KL_TR_ER &24
OUT 2211.00  ; V0416_OE_UT

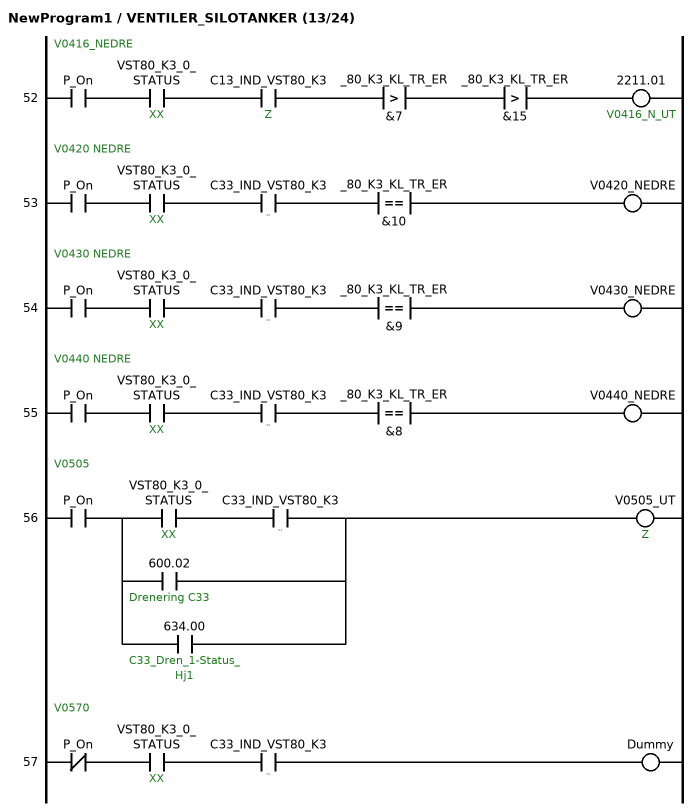
; rung 52: V0416_NEDRE
LD P_On
AND VST80_K3_0_STATUS  ; XX
AND C13_IND_VST80_K3  ; Z
AND>(320) _80_K3_KL_TR_ER &7
AND>(320) _80_K3_KL_TR_ER &15
OUT 2211.01  ; V0416_N_UT
; rung 53: V0420 NEDRE
LD P_On
AND VST80_K3_0_STATUS  ; XX
AND C33_IND_VST80_K3  ; ¨
AND=(300) _80_K3_KL_TR_ER &10
OUT V0420_NEDRE
; rung 54: V0430 NEDRE
LD P_On
AND VST80_K3_0_STATUS  ; XX
AND C33_IND_VST80_K3  ; ¨
AND=(300) _80_K3_KL_TR_ER &9
OUT V0430_NEDRE
; rung 55: V0440 NEDRE
LD P_On
AND VST80_K3_0_STATUS  ; XX
AND C33_IND_VST80_K3  ; ¨
AND=(300) _80_K3_KL_TR_ER &8
OUT V0440_NEDRE
; rung 56: V0505
LD P_On
LD VST80_K3_0_STATUS  ; XX
AND C33_IND_VST80_K3  ; ¨
OR 600.02  ; Drenering C33
OR 634.00  ; C33_Dren_1-Status_Hj1
ANDLD
OUT V0505_UT  ; Z
; rung 57: V0570
LDNOT P_On
AND VST80_K3_0_STATUS  ; XX
AND C33_IND_VST80_K3  ; ¨
OUT Dummy

